Fanuc TP program (LS listing): FOLGE123.LS

/PROG  FOLGE123
/ATTR
OWNER		= AUROM;
COMMENT		= "Posicion de Ajus";
PROG_SIZE	= 2542;
CREATE		= DATE 03-15-00  TIME 13:36:58;
MODIFIED	= DATE 24-02-18  TIME 07:17:10;
FILE_NAME	= ;
VERSION		= 0;
LINE_COUNT	= 10;
MEMORY_SIZE	= 5046;
PROTECT		= READ_WRITE;
TCD:  STACK_SIZE	= 500,
      TASK_PRIORITY	= 50,
      TIME_SLICE	= 0,
      BUSY_LAMP_OFF	= 0,
      ABORT_REQUEST	= 0,
      PAUSE_REQUEST	= 0;
DEFAULT_GROUP	= 1,1,1,1,*;
CONTROL_CODE	= 00000000 00000000;
/MN
   1:  UTOOL_NUM=24 ;
   2:  UFRAME_NUM=0 ;
   3:  PAYLOAD[1] ;
   4:J P[1] 10% CNT0 ACC100 TB   0.00sec,P-SPS    ;
      1:  IF (DO[12]=ON),CALL MAKRO998 ;
      2:  DO[15]=ON ;
      3:  DO[16]=ON ;
      4:  CALL MAKRO000    ;
      5:  WAIT (DI[9])    ;
       ------ ;
   5:J P[2] 100% CNT0 ACC100 TB   0.00sec,P-SPS    ;
      1:  TC_ONLINE (ON) ;
      2:  DO[23]=OFF ;
      3:  CALL MAKRO050    ;
      4:  DO[15]=OFF ;
      5:  WAIT (DI[23])    ;
      6:  DO[23]=ON ;
      7:  TC_ONLINE (M[30]) ;
       ------ ;
   6:J P[3] 100% CNT0 ACC100 TB    .10sec,P-SPS    ;
      1:  TC_ONLINE (ON) ;
      2:  DO[23]=OFF ;
      3:  WAIT (DI[23])    ;
      4:  DO[23]=ON ;
      5:  TC_ONLINE (M[30]) ;
       ------ ;
   7:  !Posicion de Ajuste Ejes 1-6 ;
   8:J P[4] 100% CNT0 ACC100 TB    .10sec,P-SPS    ;
      1:  TC_ONLINE (ON) ;
      2:  DO[23]=OFF ;
      3:  DO[17]=ON ;
      4:  WAIT (DI[17])    ;
      5:  DO[17]=OFF ;
      6:  WAIT (DI[23])    ;
      7:  DO[23]=ON ;
      8:  TC_ONLINE (M[30]) ;
       ------ ;
   9:J P[5] 100% CNT0 ACC100 TB    .10sec,P-SPS    ;
      1:  TC_ONLINE (ON) ;
      2:  DO[23]=OFF ;
      3:  WAIT (DI[23])    ;
      4:  DO[23]=ON ;
      5:  TC_ONLINE (M[30]) ;
       ------ ;
  10:J P[6] 100% CNT0 ACC100 TB   0.00sec,P-SPS    ;
      1:  TC_ONLINE (ON) ;
      2:  DO[14]=ON ;
      3:  DO[15]=ON ;
       ------ ;
/POS
P[1]{
   GP1:
	UF : 0, UT : 24,		CONFIG : 'F U T, 0, 1, 0',
	X =   979.595  mm,	Y =      .604  mm,	Z =   818.437  mm,
	W =  -176.060 deg,	P =    33.147 deg,	R =  -172.829 deg
   GP2:
	UF : 0, UT : 24,
	J1=   300.000  mm
   GP3:
	UF : 0, UT : 24,
	J1=     0.000  mm
   GP4:
	UF : 0, UT : 24,
	J1=     0.000  mm
};
P[2]{
   GP1:
	UF : 0, UT : 24,		CONFIG : 'F U T, 0, 1, 0',
	X =   979.595  mm,	Y =      .603  mm,	Z =   818.437  mm,
	W =  -176.060 deg,	P =    33.147 deg,	R =  -172.829 deg
   GP2:
	UF : 0, UT : 24,
	J1=   300.000  mm
   GP3:
	UF : 0, UT : 24,
	J1=     0.000  mm
   GP4:
	UF : 0, UT : 24,
	J1=     0.000  mm
};
P[3]{
   GP1:
	UF : 0, UT : 24,
	J1=    35.130 deg,	J2=   -43.479 deg,	J3=      .384 deg,
	J4=   180.033 deg,	J5=    57.088 deg,	J6=     5.946 deg
   GP2:
	UF : 0, UT : 24,
	J1=   296.600  mm
   GP3:
	UF : 0, UT : 24,
	J1=     0.000  mm
   GP4:
	UF : 0, UT : 24,
	J1=     0.000  mm
};
P[4]{
   GP1:
	UF : 0, UT : 24,
	J1=    35.135 deg,	J2=    50.149 deg,	J3=    -8.298 deg,
	J4=   180.030 deg,	J5=    71.314 deg,	J6=     5.949 deg
   GP2:
	UF : 0, UT : 24,
	J1=   295.200  mm
   GP3:
	UF : 0, UT : 24,
	J1=     0.000  mm
   GP4:
	UF : 0, UT : 24,
	J1=     0.000  mm
};
P[5]{
   GP1:
	UF : 0, UT : 24,
	J1=    35.130 deg,	J2=   -43.479 deg,	J3=      .384 deg,
	J4=   180.033 deg,	J5=    57.088 deg,	J6=     5.946 deg
   GP2:
	UF : 0, UT : 24,
	J1=   296.600  mm
   GP3:
	UF : 0, UT : 24,
	J1=     0.000  mm
   GP4:
	UF : 0, UT : 24,
	J1=     0.000  mm
};
P[6]{
   GP1:
	UF : 0, UT : 24,		CONFIG : 'F U T, 0, 1, 0',
	X =   979.595  mm,	Y =      .604  mm,	Z =   818.437  mm,
	W =  -176.060 deg,	P =    33.147 deg,	R =  -172.829 deg
   GP2:
	UF : 0, UT : 24,
	J1=   300.000  mm
   GP3:
	UF : 0, UT : 24,
	J1=     0.000  mm
   GP4:
	UF : 0, UT : 24,
	J1=     0.000  mm
};
/END
